Fanuc KAREL source: kt00380.KL

-- PROVISIONAL review KL for V770-1; original PC SHA256 09ecda70017db99d83603d7be4b212da5b5403da4008710983a8d2496aff4b1f
-- Incomplete behavior may be omitted. Consult companion uncertainty JSON. Do not deploy.
PROGRAM KT00380
%NOLOCKGROUP
VAR
  R2 : REAL
  OUT : BOOLEAN
-- UNRESOLVED_DECL H1 type=002017
BEGIN
  -- UNRESOLVED_PC offsets 5-19; opcodes 2E,22,9D,33,B4
  -- UNRESOLVED_PC offsets 24-35; opcodes 2E,23
  -- UNRESOLVED_PC offsets 40-65; opcodes 22,9D,33,B3,21,29,64,29,70,23
  -- UNRESOLVED_PC offsets 70-74; opcodes 7F
END KT00380
